FUNCTION_BLOCK PLANE_OFFSET
  (* Standard: 61499-2 *)
  (* Version 1.0, GASR *)
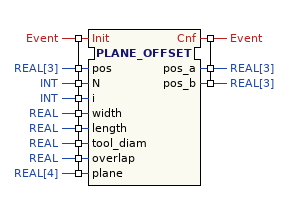
  EVENT_INPUT
    Init WITH pos, N, i, width, length, plane, tool_diam, overlap;
  END_EVENT
  EVENT_OUTPUT
    Cnf WITH pos_a, pos_b;
  END_EVENT
  VAR_INPUT
    pos : ARRAY [0..2] OF REAL;
    N : INT;
    i : INT;
    width : REAL;
    length : REAL;
    tool_diam : REAL;
    overlap : REAL;
    plane : ARRAY [0..3] OF REAL;
  END_VAR
  VAR_OUTPUT
    pos_a : ARRAY [0..2] OF REAL;
    pos_b : ARRAY [0..2] OF REAL;
  END_VAR
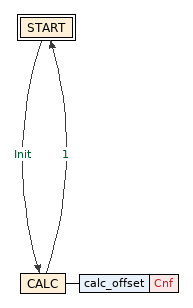
  EC_STATES
    START;
    CALC : calc_offset -> Cnf;
  END_STATES
  EC_TRANSITIONS
    CALC TO START := 1;
    START TO CALC := Init;
  END_TRANSITIONS
  ALGORITHM calc_offset IN Lua:
pos_a = {pos[1], pos[2], pos[3]}
local offx, offy, zoff
if i ~=0 then
	if length > width then
		offx = tool_diam - overlap
		offy = offx*(width - tool_diam +overlap)/(length - tool_diam +overlap)
	else
		offy = tool_diam - overlap
		offx = offy*(length - tool_diam +overlap)/(width - tool_diam +overlap)
	end
	zoff = (plane[4] - plane[2]*(pos[2]+offy) - plane[1]*(pos[1]+offx))/plane[3]
else
	offx = 0
	offy = 0
	zoff = pos[3]
end

pos_b = {pos[1] + offx, pos[2] + offy, zoff}
  END_ALGORITHM
END_FUNCTION_BLOCK
